// TwinCAT 3 PLC project PLC1_AssemblyLine
// Title: PLC1_AssemblyLine
// Company: Beckhoff Automation GmbH
// ProjectVersion: 1.0.0.0
// ProgramVersion: 3.1.4020.10
// libraries:
//   Tc2_MC2, * (Beckhoff Automation GmbH)
//   Tc2_Standard, * (Beckhoff Automation GmbH)
//   Tc2_System, * (Beckhoff Automation GmbH)
//   Tc3_EventLogger, * (Beckhoff Automation GmbH)
//   Tc3_Module, * (Beckhoff Automation GmbH)
// project tree:
//   DUTs/ E_FeederAutoState.TcDUT, E_AxisMode.TcDUT, E_StationState.TcDUT, ST_HmiAxisInfo.TcDUT, ST_HmiFeederInfo.TcDUT, ST_Hmi.TcDUT, ST_HmiAutomaticMode.TcDUT, ST_HmiErrorSimulation.TcDUT, ST_HmiFeederRecipe.TcDUT, ST_HmiManualMode.TcDUT, ST_HmiRecipeManagement.TcDUT, ST_PlcFeeder.TcDUT
//   GVLs/ GVL.TcGVL
//   / PlcTask.TcTTO
//   POUs/ FB_Axis.TcPOU, FB_Feeder.TcPOU, MAIN.TcPOU
//   Version/ Global_Version.TcGVL
// real-time tasks:
//   TASK PlcTask: cycle T#10ms, priority 10, ADS port 350
//   TASK Task 6: cycle T#10ms, priority 8, ADS port 301
// motion (NC):
//   TASK NC-Task-SAF: cycle T#2ms, priority 4, ADS port 501
//   TASK NC-Task-SVB: cycle T#10ms, priority 12, ADS port 511
//   AXIS Feeder1_AxisX (id 1)
//     OtherSettings: AllowMotionCmdToSlave=true
//     encoder EncType=1
//       SoftEndMinControl: Enable=true
//       SoftEndMaxControl: Enable=true, Range=5000
//     drive DrvType=5
//       TimeComp: TaskDelayCycles=1
//     controller CtrType=1
//       CtrPara: PriorControlFactor=1
//         Observer: BandWidth=20
//   AXIS Feeder1_AxisY (id 2)
//     OtherSettings: AllowMotionCmdToSlave=true
//     encoder EncType=1
//       SoftEndMinControl: Enable=true
//       SoftEndMaxControl: Enable=true, Range=5000
//     drive DrvType=5
//       TimeComp: TaskDelayCycles=1
//     controller CtrType=1
//       CtrPara: PriorControlFactor=1
//         Observer: BandWidth=20
//   AXIS Feeder2_AxisX (id 3)
//     OtherSettings: AllowMotionCmdToSlave=true
//     encoder EncType=1
//       SoftEndMinControl: Enable=true
//       SoftEndMaxControl: Enable=true, Range=5000
//     drive DrvType=5
//       TimeComp: TaskDelayCycles=1
//     controller CtrType=1
//       CtrPara: PriorControlFactor=1
//         Observer: BandWidth=20
//   AXIS Feeder2_AxisY (id 4)
//     OtherSettings: AllowMotionCmdToSlave=true
//     encoder EncType=1
//       SoftEndMinControl: Enable=true
//       SoftEndMaxControl: Enable=true, Range=5000
//     drive DrvType=5
//       TimeComp: TaskDelayCycles=1
//     controller CtrType=1
//       CtrPara: PriorControlFactor=1
//         Observer: BandWidth=20
// I/O:
//   DEVICE Gerät 3 (EtherCAT), AmsNetId 192.168.1.77.4.1
//     Klemme 1 (EK1100) [EK1100 EtherCAT-Koppler (2A E-Bus)]
//       Klemme 2 (EL1809) [EL1809 16K. Dig. Eingang 24V, 3ms]
//       Klemme 3 (EL2809) [EL2809 16K. Dig. Ausgang 24V, 0.5A]
//       Klemme 4 (EL9011) [EL9011 Endklemme]
// variable links:
//   PLC1_AssemblyLine/PLC1_AssemblyLine Instance <-> NC-Task-SAF/Axes/Feeder1_AxisX
//     PlcTask Inputs/MAIN.fbFeeder1.stPlcFeeder.fbAxisX.stAxis.NcToPlc <-> Outputs/ToPlc
//     PlcTask Outputs/MAIN.fbFeeder1.stPlcFeeder.fbAxisX.stAxis.PlcToNc <-> Inputs/FromPlc
//   PLC1_AssemblyLine/PLC1_AssemblyLine Instance <-> NC-Task-SAF/Axes/Feeder1_AxisY
//     PlcTask Inputs/MAIN.fbFeeder1.stPlcFeeder.fbAxisY.stAxis.NcToPlc <-> Outputs/ToPlc
//     PlcTask Outputs/MAIN.fbFeeder1.stPlcFeeder.fbAxisY.stAxis.PlcToNc <-> Inputs/FromPlc
//   PLC1_AssemblyLine/PLC1_AssemblyLine Instance <-> NC-Task-SAF/Axes/Feeder2_AxisX
//     PlcTask Inputs/MAIN.fbFeeder2.stPlcFeeder.fbAxisX.stAxis.NcToPlc <-> Outputs/ToPlc
//     PlcTask Outputs/MAIN.fbFeeder2.stPlcFeeder.fbAxisX.stAxis.PlcToNc <-> Inputs/FromPlc
//   PLC1_AssemblyLine/PLC1_AssemblyLine Instance <-> NC-Task-SAF/Axes/Feeder2_AxisY
//     PlcTask Inputs/MAIN.fbFeeder2.stPlcFeeder.fbAxisY.stAxis.NcToPlc <-> Outputs/ToPlc
//     PlcTask Outputs/MAIN.fbFeeder2.stPlcFeeder.fbAxisY.stAxis.PlcToNc <-> Inputs/FromPlc
//   Task 6 <-> Device 3 (EtherCAT)/Term 1 (EK1100)/Term 2 (EL1809)
//     Inputs/Var 1881 <-> Channel 1/Input

CONFIGURATION PLC1_AssemblyLine
    RESOURCE PLC ON TwinCAT3
        TASK PlcTask(INTERVAL := T#10ms, PRIORITY := 8);
        PROGRAM MAIN WITH PlcTask : MAIN;
    END_RESOURCE
END_CONFIGURATION

// ---- DUTs/E_FeederAutoState.TcDUT
{attribute 'qualified_only'}
TYPE E_FeederAutoState :
(
	eReset					:= 0,
	eMoveBackUp				:= 1,
	eMoveBackward			:= 2,
	eMoveDownForDragging	:= 3,
	eDrag					:= 4,
	eMoveUp					:= 5,
	eMoveForward			:= 6,
	eMoveDownForDropping	:= 7,
	eDrop					:= 8
);
END_TYPE

// ---- DUTs/E_AxisMode.TcDUT
{attribute 'qualified_only'}
TYPE E_AxisMode :
(
	INIT,
	ENABLE,
	JOG,
	POSITIONING,
	STOP,
	RESET,
	ERROR
);
END_TYPE

// ---- DUTs/E_StationState.TcDUT
{attribute 'qualified_only'}
TYPE E_StationState :
(
	eAuto	:= 2,
	eManual := 1,
	eStop	:= 0	
);
END_TYPE

// ---- DUTs/ST_HmiAxisInfo.TcDUT
TYPE ST_HmiAxisInfo :
STRUCT
	//Actual position
	fActPosition	: LREAL;
	//Actual velocity
	fActVelocity	: LREAL;
	//Current state of axis
	nAxisState		: UDINT;
	//Current mode of axis
	eAxisMode		: E_AxisMode;
END_STRUCT
END_TYPE

// ---- DUTs/ST_HmiFeederInfo.TcDUT
TYPE ST_HmiFeederInfo :
STRUCT
	//Bundled information about axis X
	stAxisX				: ST_HmiAxisInfo;
	
	//Bundled information about axis Y
	stAxisY				: ST_HmiAxisInfo;
	
	//Information about the gripper
	bGripperIsClosed	: BOOL;
END_STRUCT
END_TYPE

// ---- DUTs/ST_Hmi.TcDUT
TYPE ST_Hmi :
STRUCT
	//Operation mode 
	nStationState_Request	: INT;
	nStationState_Respond	: INT;	
	
	//Bundled manual mode settings and feedback
	stManualMode			: ST_HmiManualMode;
	
	//Bundled automatic mode settings and feedback
	stAutomaticMode			: ST_HmiAutomaticMode;
	
	//Bundled teach mode / recipe management settings and feedback
	stRecipeManagement		: ST_HmiRecipeManagement;
	
	//Bundled error simulation
	stErrorSimulation		: ST_HmiErrorSimulation;
	
	//Bundled feeder information
	stFeederInfo			: ST_HmiFeederInfo;
END_STRUCT
END_TYPE

// ---- DUTs/ST_HmiAutomaticMode.TcDUT
TYPE ST_HmiAutomaticMode :
STRUCT
	//Current state of the automatic mode state machine
	nStateNumber		: INT := 0;
END_STRUCT
END_TYPE

// ---- DUTs/ST_HmiErrorSimulation.TcDUT
TYPE ST_HmiErrorSimulation :
STRUCT
	bOnMoveBackUp			: BOOL;
	bOnMoveBackward			: BOOL;
	bOnMoveDownForDragging	: BOOL;
	bOnDrag					: BOOL;
	bOnMoveUp				: BOOL;
	bOnMoveForward			: BOOL;
	bOnMoveDownForDropping	: BOOL;
	bOnDrop					: BOOL;
END_STRUCT
END_TYPE

// ---- DUTs/ST_HmiFeederRecipe.TcDUT
TYPE ST_HmiFeederRecipe :
STRUCT
	//Target 1 name
	sTarget1Name			: STRING := 'Target Pos1';
	//Target 1 positon for X axis
	fTarget1PositionX		: LREAL	:= LREAL#0.0;
	//Target 1 position for Y axis
	fTarget1PositionY		: LREAL	:= LREAL#0.0;

	//Target 2 name
	sTarget2Name			: STRING := 'Target Pos2';
	//Target 2 positon for X axis
	fTarget2PositionX		: LREAL	:= LREAL#1000.0;
	//Target 2 position for Y axis
	fTarget2PositionY		: LREAL	:= LREAL#2000.0;
	
	//Velocity of both axis	
	fVelocity				: LREAL := 500;
END_STRUCT
END_TYPE

// ---- DUTs/ST_HmiManualMode.TcDUT
TYPE ST_HmiManualMode :
STRUCT
	//Manual mode - move X axis forward
	bButtonForwardX			: BOOL;
	//Manual mode - move X axis backward
	bButtonBackwardX		: BOOL;
	//Manual mode - move Y axis forward
	bButtonForwardY		: BOOL;
	//Manual mode - move Y axis backward
	bButtonBackwardY		: BOOL;
	//Manual mode - close gripper
	bButtonCloseGripper		: BOOL;
	//Manual mode - velocity X axis	
	fVelocityX			: LREAL := 500;
	//Manual mode - velocity Y axis
	fVelocityY			: LREAL := 500;
END_STRUCT
END_TYPE

// ---- DUTs/ST_HmiRecipeManagement.TcDUT
TYPE ST_HmiRecipeManagement :
STRUCT
	//Current recipe name
	sCurrentRecipeName	: STRING(50)	:= 'Unknown recipe';

	//Feeder recipe data
	stFeederRecipe		: ST_HmiFeederRecipe;
END_STRUCT
END_TYPE

// ---- DUTs/ST_PlcFeeder.TcDUT
TYPE ST_PlcFeeder :
STRUCT
	//ID of the feeder as identification in hmi, log, etc.
	nFeederId				: USINT;

	//Current operation mode of the machine
	eStationState			: E_StationState;
	
	//Delay for simulating drag and drop
	fbTonAuto				: TON;
	
	//State machine of automatic mode
	eAutoState				: E_FeederAutoState;

	//NC-drive X axis
	fbAxisX					: FB_Axis;
	//NC-drive Y axis
	fbAxisY					: FB_Axis;	

	//Gripper status
	bCloseGripper			: BOOL;
	bGripperIsClosed		: BOOL;
	
	//Current position of the X axis for historize extension in the HMI server
	fHmiPosXHistorize		: LREAL;
	//Current position of the Y axis for historize extension in the HMI server
	fHmiPosYHistorize		: LREAL;
	//Current velocity of the X axis for historize extension in the HMI server
	fHmiVeloXHistorize		: LREAL;
	//Current velocity of the Y axis for historize extension in the HMI server
	fHmiVeloYHistorize		: LREAL;
	
END_STRUCT
END_TYPE

// ---- GVLs/GVL.TcGVL
{attribute 'qualified_only'}
VAR_GLOBAL
	bAxisError	: BOOL;
END_VAR

// ---- Version/Global_Version.TcGVL
{attribute 'TcGenerated'}
// This function has been automatically generated from the project information.
VAR_GLOBAL CONSTANT
	{attribute 'const_non_replaced'}
	{attribute 'linkalways'}
	stLibVersion_PLC1_AssemblyLine : ST_LibVersion := (iMajor := 1, iMinor := 0, iBuild := 0, iRevision := 0, sVersion := '1.0.0.0');
END_VAR

// ---- POUs/MAIN.TcPOU
PROGRAM MAIN
VAR
	fbFeeder1		: FB_Feeder(nFeederId := 1);
	fbFeeder2		: FB_Feeder(nFeederId := 2);
END_VAR

fbFeeder1();
fbFeeder2();

END_PROGRAM

// ---- POUs/FB_Feeder.TcPOU
FUNCTION_BLOCK FB_Feeder
VAR_INPUT
END_VAR
VAR_OUTPUT
END_VAR
VAR
	
	stPlcFeeder				: ST_PlcFeeder;
	
	//Struct for communication with the HMI
	stHmi					: ST_Hmi;
END_VAR
VAR PERSISTENT
	//Current target positions from hmi recipe management
	stTargets				: ST_HmiFeederRecipe;
END_VAR

// Drives
stPlcFeeder.fbAxisX();
stPlcFeeder.fbAxisY();

// Hmi
M_Hmi();

// state machine
M_StationState();

// Events
M_Events();

CASE stHmi.nStationState_Request OF
	0: stPlcFeeder.eStationState := E_StationState.eStop;
	1: stPlcFeeder.eStationState := E_StationState.eManual;
	2: stPlcFeeder.eStationState := E_StationState.eAuto;
END_CASE

METHOD FB_init : BOOL
VAR_INPUT
	bInitRetains	: BOOL; // if TRUE, the retain variables are initialized (warm start / cold start)
	bInCopyCode		: BOOL;  // if TRUE, the instance afterwards gets moved into the copy code (online change)
	nFeederId		: USINT;
END_VAR
FeederId := nFeederId;
END_METHOD

PROPERTY PUBLIC FeederId : USINT
GET // PUBLIC
FeederId := stPlcFeeder.nFeederId;
END_GET
SET // PRIVATE
stPlcFeeder.nFeederId := FeederId;
END_SET
END_PROPERTY

METHOD M_Auto
VAR_INPUT
END_VAR
// Stoppping all axis for op mode change
IF stHmi.nStationState_Request <> 2 THEN
	stPlcFeeder.fbAxisX.bInStop := TRUE;
	stPlcFeeder.fbAxisY.bInStop := TRUE;
	RETURN;
END_IF

stPlcFeeder.fbTonAuto();
stPlcFeeder.fbAxisX.fInOverride := LREAL#100;    
stPlcFeeder.fbAxisX.fInVelocity := stTargets.fVelocity;
stPlcFeeder.fbAxisY.fInOverride := LREAL#100;    
stPlcFeeder.fbAxisY.fInVelocity := stTargets.fVelocity;

// State machine automatic mode
CASE stPlcFeeder.eAutoState OF
	E_FeederAutoState.eReset:
		M_AutoReset();
	E_FeederAutoState.eMoveBackUp:
		M_AutoMoveBackUp();
	E_FeederAutoState.eMoveBackward:
		M_AutoMoveBackward();	
	E_FeederAutoState.eMoveDownForDragging:
		M_AutoMoveDownForDragging();
	E_FeederAutoState.eDrag:
		M_AutoDrag();
	E_FeederAutoState.eMoveUp:
		M_AutoMoveUp();
	E_FeederAutoState.eMoveForward:
		M_AutoMoveForward();
	E_FeederAutoState.eMoveDownForDropping:
		M_AutoMoveDownForDropping();
	E_FeederAutoState.eDrop:
		M_AutoDrop();	
END_CASE
END_METHOD

METHOD M_AutoDrag
VAR_INPUT
END_VAR
VAR_INST
	fbAlarm						: Tc3_EventLogger.FB_TcAlarm;
	bWaitForErrorConfirmation	: BOOL;
	bConfirmManualy				: BOOL;
END_VAR
IF stHmi.stErrorSimulation.bOnDrag THEN
	fbAlarm.CreateEx(TC_EVENTS.AssemblyLineEvents.AutomaticModeError, TRUE, 0);
	fbAlarm.ipArguments.Clear().AddInt(stPlcFeeder.eAutoState);
END_IF

IF NOT bWaitForErrorConfirmation THEN
	stPlcFeeder.fbTonAuto.PT := T#2S;
	stPlcFeeder.fbTonAuto.IN := TRUE;
	stPlcFeeder.bCloseGripper := TRUE;
END_IF

IF stPlcFeeder.fbTonAuto.Q THEN
	stPlcFeeder.fbTonAuto.IN := FALSE;
	IF stHmi.stErrorSimulation.bOnDrag THEN
		stHmi.stErrorSimulation.bOnDrag := FALSE;		
		fbAlarm.Raise(0);
		bWaitForErrorConfirmation := TRUE;
	ELSE
		stPlcFeeder.bGripperIsClosed := TRUE;
		stPlcFeeder.eAutoState := E_FeederAutoState.eMoveUp;
	END_IF		
END_IF

IF bWaitForErrorConfirmation AND fbAlarm.eConfirmationState = TcEventConfirmationState.Confirmed THEN
	bWaitForErrorConfirmation := FALSE;
	fbAlarm.Clear(0,TRUE);	
	stPlcFeeder.bGripperIsClosed := TRUE;
	stPlcFeeder.eAutoState := E_FeederAutoState.eMoveUp;
END_IF

IF bConfirmManualy THEN
	bConfirmManualy := FALSE;
	fbAlarm.Confirm(0);
END_IF
END_METHOD

METHOD M_AutoDrop
VAR_INPUT
END_VAR
VAR_INST
	fbAlarm						: Tc3_EventLogger.FB_TcAlarm;
	bWaitForErrorConfirmation	: BOOL;
	bConfirmManualy				: BOOL;
END_VAR
IF stHmi.stErrorSimulation.bOnDrop THEN
	fbAlarm.CreateEx(TC_EVENTS.AssemblyLineEvents.AutomaticModeError, TRUE, 0);
	fbAlarm.ipArguments.Clear().AddInt(stPlcFeeder.eAutoState);
END_IF

IF NOT bWaitForErrorConfirmation THEN
	stPlcFeeder.fbTonAuto.PT := T#2S;
	stPlcFeeder.fbTonAuto.IN := TRUE;
	stPlcFeeder.bCloseGripper := FALSE;
END_IF

IF stPlcFeeder.fbTonAuto.Q THEN
	stPlcFeeder.fbTonAuto.IN := FALSE;
	IF stHmi.stErrorSimulation.bOnDrop THEN
		stHmi.stErrorSimulation.bOnDrop := FALSE;		
		fbAlarm.Raise(0);
		bWaitForErrorConfirmation := TRUE;
	ELSE
		stPlcFeeder.bGripperIsClosed := FALSE;
		stPlcFeeder.eAutoState := E_FeederAutoState.eMoveBackUp;
	END_IF		
END_IF

IF bWaitForErrorConfirmation AND fbAlarm.eConfirmationState = TcEventConfirmationState.Confirmed THEN
	bWaitForErrorConfirmation := FALSE;	
	fbAlarm.Clear(0,TRUE);
	stPlcFeeder.bGripperIsClosed := FALSE;
	stPlcFeeder.eAutoState := E_FeederAutoState.eMoveBackUp;
END_IF

IF bConfirmManualy THEN
	bConfirmManualy := FALSE;
	fbAlarm.Confirm(0);
END_IF
END_METHOD

METHOD M_AutoMoveBackUp
VAR_INPUT
END_VAR
VAR_INST
	fbAlarm						: Tc3_EventLogger.FB_TcAlarm;
	bWaitForErrorConfirmation	: BOOL;
	bConfirmManualy				: BOOL;
END_VAR
IF stHmi.stErrorSimulation.bOnMoveBackUp THEN
	fbAlarm.CreateEx(TC_EVENTS.AssemblyLineEvents.AutomaticModeError, TRUE, 0);
	fbAlarm.ipArguments.Clear().AddInt(stPlcFeeder.eAutoState);
END_IF

stPlcFeeder.fbAxisY.fInTargetPos := 0.0;

IF stPlcFeeder.fbAxisY.fOutActPosition <> 0 THEN
	stPlcFeeder.fbAxisY.bInPositioning := TRUE;
	IF stHmi.stErrorSimulation.bOnMoveBackUp THEN
		stHmi.stErrorSimulation.bOnMoveBackUp := FALSE;
		stPlcFeeder.fbAxisX.bInPositioning := FALSE;		
		stPlcFeeder.fbAxisY.bInPositioning := FALSE;		
		stPlcFeeder.fbAxisX.bInStop := TRUE;
		stPlcFeeder.fbAxisY.bInStop := TRUE;
		fbAlarm.Raise(0);
		bWaitForErrorConfirmation := TRUE;
	END_IF
ELSIF stPlcFeeder.fbAxisY.fOutActPosition = 0 AND NOT bWaitForErrorConfirmation THEN 
	stPlcFeeder.fbAxisY.bInPositioning := FALSE;
	stPlcFeeder.eAutoState :=  E_FeederAutoState.eMoveBackward;
END_IF

IF bWaitForErrorConfirmation AND fbAlarm.eConfirmationState = TcEventConfirmationState.Confirmed THEN
	bWaitForErrorConfirmation := FALSE;	
	fbAlarm.Clear(0,TRUE);
	stPlcFeeder.fbAxisX.bInStop := FALSE;
	stPlcFeeder.fbAxisY.bInStop := FALSE;
	stPlcFeeder.fbAxisY.bInPositioning := TRUE;
END_IF

IF bConfirmManualy THEN
	bConfirmManualy := FALSE;
	fbAlarm.Confirm(0);
END_IF
END_METHOD

METHOD M_AutoMoveBackward
VAR_INPUT
END_VAR
VAR_INST
	fbAlarm						: Tc3_EventLogger.FB_TcAlarm;
	bWaitForErrorConfirmation	: BOOL;
	bConfirmManualy				: BOOL;
END_VAR
IF stHmi.stErrorSimulation.bOnMoveBackward THEN
	fbAlarm.CreateEx(TC_EVENTS.AssemblyLineEvents.AutomaticModeError, TRUE, 0);
	fbAlarm.ipArguments.Clear().AddInt(stPlcFeeder.eAutoState);
END_IF

stPlcFeeder.fbAxisX.fInTargetPos := stTargets.fTarget1PositionX;

IF stPlcFeeder.fbAxisX.fOutActPosition <> stTargets.fTarget1PositionX THEN
	stPlcFeeder.fbAxisX.bInPositioning := TRUE;
	IF stHmi.stErrorSimulation.bOnMoveBackward THEN
		stHmi.stErrorSimulation.bOnMoveBackward := FALSE;
		stPlcFeeder.fbAxisX.bInPositioning := FALSE;		
		stPlcFeeder.fbAxisY.bInPositioning := FALSE;		
		stPlcFeeder.fbAxisX.bInStop := TRUE;
		stPlcFeeder.fbAxisY.bInStop := TRUE;
		fbAlarm.Raise(0);
		bWaitForErrorConfirmation := TRUE;
	END_IF
ELSIF stPlcFeeder.fbAxisX.fOutActPosition = stTargets.fTarget1PositionX AND NOT bWaitForErrorConfirmation THEN 
	stPlcFeeder.fbAxisX.bInPositioning := FALSE;
	stPlcFeeder.eAutoState := E_FeederAutoState.eMoveDownForDragging;
END_IF

IF bWaitForErrorConfirmation AND fbAlarm.eConfirmationState = TcEventConfirmationState.Confirmed THEN
	bWaitForErrorConfirmation := FALSE;	
	fbAlarm.Clear(0,TRUE);	
	stPlcFeeder.fbAxisX.bInStop := FALSE;
	stPlcFeeder.fbAxisY.bInStop := FALSE;
	stPlcFeeder.fbAxisX.bInPositioning := TRUE;
END_IF

IF bConfirmManualy THEN
	bConfirmManualy := FALSE;
	fbAlarm.Confirm(0);
END_IF
END_METHOD

METHOD M_AutoMoveDownForDragging
VAR_INPUT
END_VAR
VAR_INST
	fbAlarm						: Tc3_EventLogger.FB_TcAlarm;
	bWaitForErrorConfirmation	: BOOL;
	bConfirmManualy				: BOOL;
END_VAR
IF stHmi.stErrorSimulation.bOnMoveDownForDragging THEN
	fbAlarm.CreateEx(TC_EVENTS.AssemblyLineEvents.AutomaticModeError, TRUE, 0);
	fbAlarm.ipArguments.Clear().AddInt(stPlcFeeder.eAutoState);
END_IF

stPlcFeeder.fbAxisY.fInTargetPos := stTargets.fTarget1PositionY;

IF stPlcFeeder.fbAxisY.fOutActPosition <> stTargets.fTarget1PositionY THEN
	stPlcFeeder.fbAxisY.bInPositioning := TRUE;
	IF stHmi.stErrorSimulation.bOnMoveDownForDragging THEN
		stHmi.stErrorSimulation.bOnMoveDownForDragging := FALSE;
		stPlcFeeder.fbAxisX.bInPositioning := FALSE;		
		stPlcFeeder.fbAxisY.bInPositioning := FALSE;		
		stPlcFeeder.fbAxisX.bInStop := TRUE;
		stPlcFeeder.fbAxisY.bInStop := TRUE;
		fbAlarm.Raise(0);
		bWaitForErrorConfirmation := TRUE;
	END_IF
ELSIF stPlcFeeder.fbAxisY.fOutActPosition = stTargets.fTarget1PositionY AND NOT bWaitForErrorConfirmation THEN 
	stPlcFeeder.fbAxisY.bInPositioning := FALSE;
	stPlcFeeder.eAutoState := E_FeederAutoState.eDrag;
END_IF

IF bWaitForErrorConfirmation AND fbAlarm.eConfirmationState = TcEventConfirmationState.Confirmed THEN
	bWaitForErrorConfirmation := FALSE;	
	fbAlarm.Clear(0,TRUE);
	stPlcFeeder.fbAxisX.bInStop := FALSE;
	stPlcFeeder.fbAxisY.bInStop := FALSE;
	stPlcFeeder.fbAxisY.bInPositioning := TRUE;
END_IF

IF bConfirmManualy THEN
	bConfirmManualy := FALSE;
	fbAlarm.Confirm(0);
END_IF
END_METHOD

METHOD M_AutoMoveDownForDropping
VAR_INPUT
END_VAR
VAR_INST
	fbAlarm						: Tc3_EventLogger.FB_TcAlarm;
	bWaitForErrorConfirmation	: BOOL;
	bConfirmManualy				: BOOL;
END_VAR
IF stHmi.stErrorSimulation.bOnMoveDownForDropping THEN
	fbAlarm.CreateEx(TC_EVENTS.AssemblyLineEvents.AutomaticModeError, TRUE, 0);
	fbAlarm.ipArguments.Clear().AddInt(stPlcFeeder.eAutoState);
END_IF

stPlcFeeder.fbAxisY.fInTargetPos := stTargets.fTarget2PositionY;

IF stPlcFeeder.fbAxisY.fOutActPosition <> stTargets.fTarget2PositionY THEN
	stPlcFeeder.fbAxisY.bInPositioning := TRUE;
	IF stHmi.stErrorSimulation.bOnMoveDownForDropping THEN
		stHmi.stErrorSimulation.bOnMoveDownForDropping := FALSE;
		stPlcFeeder.fbAxisX.bInPositioning := FALSE;		
		stPlcFeeder.fbAxisY.bInPositioning := FALSE;		
		stPlcFeeder.fbAxisX.bInStop := TRUE;
		stPlcFeeder.fbAxisY.bInStop := TRUE;
		fbAlarm.Raise(0);
		bWaitForErrorConfirmation := TRUE;
	END_IF
ELSIF stPlcFeeder.fbAxisY.fOutActPosition = stTargets.fTarget2PositionY AND NOT bWaitForErrorConfirmation THEN 
	stPlcFeeder.fbAxisY.bInPositioning := FALSE;
	stPlcFeeder.eAutoState := E_FeederAutoState.eDrop;
END_IF

IF bWaitForErrorConfirmation AND fbAlarm.eConfirmationState = TcEventConfirmationState.Confirmed THEN
	bWaitForErrorConfirmation := FALSE;	
	fbAlarm.Clear(0,TRUE);
	stPlcFeeder.fbAxisX.bInStop := FALSE;
	stPlcFeeder.fbAxisY.bInStop := FALSE;
	stPlcFeeder.fbAxisY.bInPositioning := TRUE;
END_IF

IF bConfirmManualy THEN
	bConfirmManualy := FALSE;
	fbAlarm.Confirm(0);
END_IF
END_METHOD

METHOD M_AutoMoveForward
VAR_INPUT
END_VAR
VAR_INST
	fbAlarm						: Tc3_EventLogger.FB_TcAlarm;
	bWaitForErrorConfirmation	: BOOL;
	bConfirmManualy				: BOOL;
END_VAR
IF stHmi.stErrorSimulation.bOnMoveForward THEN
	fbAlarm.CreateEx(TC_EVENTS.AssemblyLineEvents.AutomaticModeError, TRUE, 0);
	fbAlarm.ipArguments.Clear().AddInt(stPlcFeeder.eAutoState);
END_IF

stPlcFeeder.fbAxisX.fInTargetPos := stTargets.fTarget2PositionX;

IF stPlcFeeder.fbAxisX.fOutActPosition <> stTargets.fTarget2PositionX THEN
	stPlcFeeder.fbAxisX.bInPositioning := TRUE;
	IF stHmi.stErrorSimulation.bOnMoveForward THEN
		stHmi.stErrorSimulation.bOnMoveForward := FALSE;
		stPlcFeeder.fbAxisX.bInPositioning := FALSE;		
		stPlcFeeder.fbAxisY.bInPositioning := FALSE;		
		stPlcFeeder.fbAxisX.bInStop := TRUE;
		stPlcFeeder.fbAxisY.bInStop := TRUE;
		fbAlarm.Raise(0);
		bWaitForErrorConfirmation := TRUE;
	END_IF
ELSIF stPlcFeeder.fbAxisX.fOutActPosition = stTargets.fTarget2PositionX AND NOT bWaitForErrorConfirmation THEN 
	stPlcFeeder.fbAxisX.bInPositioning := FALSE;
	stPlcFeeder.eAutoState := E_FeederAutoState.eMoveDownForDropping;
END_IF

IF bWaitForErrorConfirmation AND fbAlarm.eConfirmationState = TcEventConfirmationState.Confirmed THEN
	bWaitForErrorConfirmation := FALSE;	
	fbAlarm.Clear(0,TRUE);
	stPlcFeeder.fbAxisX.bInStop := FALSE;
	stPlcFeeder.fbAxisY.bInStop := FALSE;
	stPlcFeeder.fbAxisX.bInPositioning := TRUE;
END_IF

IF bConfirmManualy THEN
	bConfirmManualy := FALSE;
	fbAlarm.Confirm(0);
END_IF
END_METHOD

METHOD M_AutoMoveUp
VAR_INPUT
END_VAR
VAR_INST
	fbAlarm						: Tc3_EventLogger.FB_TcAlarm;
	bWaitForErrorConfirmation	: BOOL;
	bConfirmManualy				: BOOL;
END_VAR
IF stHmi.stErrorSimulation.bOnMoveUp THEN
	fbAlarm.CreateEx(TC_EVENTS.AssemblyLineEvents.AutomaticModeError, TRUE, 0);
	fbAlarm.ipArguments.Clear().AddInt(stPlcFeeder.eAutoState);
END_IF

stPlcFeeder.fbAxisY.fInTargetPos := 0.0;

IF stPlcFeeder.fbAxisY.fOutActPosition <> 0 THEN
	stPlcFeeder.fbAxisY.bInPositioning := TRUE;
	IF stHmi.stErrorSimulation.bOnMoveUp THEN
		stHmi.stErrorSimulation.bOnMoveUp := FALSE;
		stPlcFeeder.fbAxisX.bInPositioning := FALSE;		
		stPlcFeeder.fbAxisY.bInPositioning := FALSE;		
		stPlcFeeder.fbAxisX.bInStop := TRUE;
		stPlcFeeder.fbAxisY.bInStop := TRUE;
		fbAlarm.Raise(0);
		bWaitForErrorConfirmation := TRUE;
	END_IF
ELSIF stPlcFeeder.fbAxisY.fOutActPosition = 0 AND NOT bWaitForErrorConfirmation THEN 
	stPlcFeeder.fbAxisY.bInPositioning := FALSE;
	stPlcFeeder.eAutoState := E_FeederAutoState.eMoveForward;
END_IF

IF bWaitForErrorConfirmation AND fbAlarm.eConfirmationState = TcEventConfirmationState.Confirmed THEN
	bWaitForErrorConfirmation := FALSE;	
	fbAlarm.Clear(0,TRUE);
	stPlcFeeder.fbAxisX.bInStop := FALSE;
	stPlcFeeder.fbAxisY.bInStop := FALSE;
	stPlcFeeder.fbAxisY.bInPositioning := TRUE;
END_IF

IF bConfirmManualy THEN
	bConfirmManualy := FALSE;
	fbAlarm.Confirm(0);
END_IF
END_METHOD

METHOD M_AutoReset
VAR_INPUT
END_VAR
stPlcFeeder.fbAxisX.fInTargetPos := 0.0;
stPlcFeeder.fbAxisY.fInTargetPos := 0.0;
stPlcFeeder.fbAxisX.bInStop := FALSE;
stPlcFeeder.fbAxisY.bInStop := FALSE;

IF stPlcFeeder.fbAxisX.fOutActPosition <> 0 THEN 
	stPlcFeeder.fbAxisX.bInPositioning := TRUE;
END_IF

IF stPlcFeeder.fbAxisY.fOutActPosition <> 0 THEN 
	stPlcFeeder.fbAxisY.bInPositioning := TRUE;
END_IF

IF stPlcFeeder.fbAxisX.fOutActPosition = 0 AND stPlcFeeder.fbAxisY.fOutActPosition = 0 THEN 
	stPlcFeeder.fbAxisX.bInPositioning := FALSE;
	stPlcFeeder.fbAxisY.bInPositioning := FALSE;
	stPlcFeeder.eAutoState := E_FeederAutoState.eMoveBackUp;
END_IF
END_METHOD

METHOD PRIVATE M_Events : BOOL
VAR_INPUT
END_VAR
VAR
	sJsonAttributeAxis		: STRING;
END_VAR
VAR_INST
	fbTriggerAutomaticOn	: R_TRIG;
	fbTriggerManualModeOn	: R_TRIG;
	fbTriggerStop			: R_TRIG;
	fbTriggerErrorAxisX		: R_TRIG;
	fbTriggerErrorAxisY		: R_TRIG;	
	fbMessage 				: Tc3_EventLogger.FB_TcMessage;
	fbAlarmAxisX			: Tc3_EventLogger.FB_TcAlarm;
	fbAlarmAxisY			: Tc3_EventLogger.FB_TcAlarm;
END_VAR
fbTriggerAutomaticOn(CLK := stPlcFeeder.eStationState = E_StationState.eAuto);
IF fbTriggerAutomaticOn.Q THEN
	fbMessage.CreateEx(TC_EVENTS.AssemblyLineEvents.FeederAutomaticOn, 0);
	fbMessage.ipArguments.Clear().AddUSInt(FeederId);
	fbMessage.Send(0);
END_IF

fbTriggerManualModeOn(CLK := stPlcFeeder.eStationState = E_StationState.eManual);
IF fbTriggerManualModeOn.Q THEN
	fbMessage.CreateEx(TC_EVENTS.AssemblyLineEvents.FeederManualModeOn, 0);
	fbMessage.ipArguments.Clear().AddUSInt(FeederId);
	fbMessage.Send(0);
END_IF

fbTriggerStop(CLK := stPlcFeeder.eStationState = E_StationState.eStop);
IF fbTriggerStop.Q THEN
	fbMessage.CreateEx(TC_EVENTS.AssemblyLineEvents.FeederStopped, 0);
	fbMessage.ipArguments.Clear().AddUSInt(FeederId);
	fbMessage.Send(0);
END_IF

fbTriggerErrorAxisX(CLK := stPlcFeeder.fbAxisX.bOutError);
IF fbTriggerErrorAxisX.Q THEN
	fbAlarmAxisX.Clear(0, TRUE);
	fbAlarmAxisX.CreateEx(TC_EVENTS.AssemblyLineEvents.FeederError, FALSE, 0);
	fbAlarmAxisX.ipArguments.Clear().AddUSInt(FeederId).AddString('X');
	sJsonAttributeAxis := CONCAT(CONCAT('{"ErrorId: ', TO_STRING(stPlcFeeder.fbAxisX.nOutErrorId)), '}');
	fbAlarmAxisX.SetJsonAttribute(sJsonAttributeAxis);
	fbAlarmAxisX.Raise(0);
END_IF

fbTriggerErrorAxisY(CLK := stPlcFeeder.fbAxisY.bOutError);
IF fbTriggerErrorAxisY.Q THEN
	fbAlarmAxisY.Clear(0, TRUE);
	fbAlarmAxisY.CreateEx(TC_EVENTS.AssemblyLineEvents.FeederError, FALSE, 0);
	fbAlarmAxisY.ipArguments.Clear().AddUSInt(FeederId).AddString('Y');
	sJsonAttributeAxis := CONCAT(CONCAT('{"ErrorId: ', TO_STRING(stPlcFeeder.fbAxisY.nOutErrorId)), '}');
	fbAlarmAxisY.SetJsonAttribute(sJsonAttributeAxis);
	fbAlarmAxisY.Raise(0);
END_IF
END_METHOD

METHOD M_Hmi : BOOL
VAR_INPUT
END_VAR
IF _TaskInfo[GETCURTASKINDEXEX()].FirstCycle THEN
	stHmi.stRecipeManagement.stFeederRecipe := stTargets;
END_IF

stHmi.nStationState_Respond := TO_INT(stPlcFeeder.eStationState);

stHmi.stAutomaticMode.nStateNumber := stPlcFeeder.eAutoState;
stHmi.stFeederInfo.bGripperIsClosed := stPlcFeeder.bGripperIsClosed;

// HMI historize actual position and velocity
stPlcFeeder.fHmiPosXHistorize := stPlcFeeder.fbAxisX.fOutActPosition;
stPlcFeeder.fHmiPosYHistorize := stPlcFeeder.fbAxisY.fOutActPosition;
stPlcFeeder.fHmiVeloXHistorize := stPlcFeeder.fbAxisX.fOutActVelocity;
stPlcFeeder.fHmiVeloYHistorize := stPlcFeeder.fbAxisY.fOutActVelocity;

// HMI axis information
stHmi.stFeederInfo.stAxisX.fActPosition := stPlcFeeder.fbAxisX.fOutActPosition;
stHmi.stFeederInfo.stAxisX.fActVelocity := stPlcFeeder.fbAxisX.fOutActVelocity;
stHmi.stFeederInfo.stAxisX.nAxisState := stPlcFeeder.fbAxisX.nOutAxisState;
stHmi.stFeederInfo.stAxisX.eAxisMode := stPlcFeeder.fbAxisX.eOutAxisMode;

stHmi.stFeederInfo.stAxisY.fActPosition := stPlcFeeder.fbAxisY.fOutActPosition;
stHmi.stFeederInfo.stAxisY.fActVelocity := stPlcFeeder.fbAxisY.fOutActVelocity;
stHmi.stFeederInfo.stAxisY.nAxisState := stPlcFeeder.fbAxisY.nOutAxisState;
stHmi.stFeederInfo.stAxisY.eAxisMode := stPlcFeeder.fbAxisY.eOutAxisMode;

//Set targets from hmi recipe management
stTargets := stHmi.stRecipeManagement.stFeederRecipe;
END_METHOD

METHOD M_Man
VAR_INPUT
END_VAR
// Stoppping all axis for op mode change
IF stHmi.nStationState_Request <> 1 THEN
	stPlcFeeder.fbAxisX.bInStop := TRUE;
	stPlcFeeder.fbAxisY.bInStop := TRUE;
	stPlcFeeder.fbAxisX.bInJog := FALSE;
	stPlcFeeder.fbAxisY.bInJog := FALSE;
	stPlcFeeder.eAutoState := E_FeederAutoState.eReset;
	RETURN;
END_IF

stPlcFeeder.fbAxisX.bInStop := FALSE;
stPlcFeeder.fbAxisX.bInJog := TRUE;
stPlcFeeder.fbAxisX.fInOverride := LREAL#100;
stPlcFeeder.fbAxisX.fInVelocity := stHmi.stManualMode.fVelocityX;
stPlcFeeder.fbAxisX.bInJogForward := stHmi.stManualMode.bButtonForwardX;
stPlcFeeder.fbAxisX.bInJogBackward := stHmi.stManualMode.bButtonBackwardX;

stPlcFeeder.fbAxisY.bInStop := FALSE;
stPlcFeeder.fbAxisY.bInJog := TRUE;
stPlcFeeder.fbAxisY.fInOverride := LREAL#100;
stPlcFeeder.fbAxisY.fInVelocity := stHmi.stManualMode.fVelocityY;
stPlcFeeder.fbAxisY.bInJogForward := stHmi.stManualMode.bButtonForwardY;
stPlcFeeder.fbAxisY.bInJogBackward := stHmi.stManualMode.bButtonBackwardY;

stPlcFeeder.bCloseGripper := stHmi.stManualMode.bButtonCloseGripper;
END_METHOD

METHOD M_StationState
VAR_INPUT
END_VAR

VAR

END_VAR
CASE stPlcFeeder.eStationState OF
	E_StationState.eAuto:
		M_Auto();
	E_StationState.eManual:
		M_Man();
	E_StationState.eStop:
		M_Stop();	
END_CASE
END_METHOD

METHOD M_Stop
VAR_INPUT
END_VAR
stPlcFeeder.fbAxisX.bInStop := TRUE;
stPlcFeeder.fbAxisY.bInStop := TRUE;

IF stHmi.nStationState_Request = 2 THEN
	stPlcFeeder.eAutoState := E_FeederAutoState.eReset;
END_IF
END_METHOD

END_FUNCTION_BLOCK

// ---- POUs/FB_Axis.TcPOU
FUNCTION_BLOCK FB_Axis
VAR_INPUT
	// Commands
	bInJog				: BOOL;
	bInJogForward		: BOOL;
	bInJogBackward		: BOOL;
	bInPositioning		: BOOL;
	bInStop				: BOOL;
	bInReset			: BOOL;

	// Parameters
	fInVelocity			: LREAL := 1000.0;
	fInOverride			: LREAL := 100;
	fInTargetPos		: LREAL := 0;	
END_VAR
VAR_OUTPUT
	// Status
	bOutError			: BOOL;
	nOutErrorId			: UDINT;
	fOutActPosition		: DINT;
	fOutActVelocity		: DINT;
	fOutSetPosition		: LREAL;
	fOutSetVelocity		: LREAL;
	nOutAxisState		: UDINT;
	eOutAxisMode		: E_AxisMode;    
END_VAR
VAR
	// MC function blocks
	fbPower			: Tc2_MC2.MC_Power;
	fbReset			: Tc2_MC2.MC_Reset;
	fbStop			: Tc2_MC2.MC_Stop;	
	fbMoveAbs		: Tc2_MC2.MC_MoveAbsolute;
	fbJog			: Tc2_MC2.MC_Jog;
	
	// MC structures	
	stAxis			: Tc2_MC2.AXIS_REF;
	stPower			: Tc2_MC2.ST_McOutputs;
	stReset			: Tc2_MC2.ST_McOutputs;
	stStop			: Tc2_MC2.ST_McOutputs;
	stMoveAbs		: Tc2_MC2.ST_McOutputs;
	stJog			: Tc2_MC2.ST_McOutputs;
	
	// state machine
	eAxisMode		: E_AxisMode;
END_VAR

stAxis.ReadStatus();

// state machine
CASE eAxisMode OF

		E_AxisMode.INIT:
		
					fbPower.Enable := FALSE;
					fbReset.Execute := FALSE;
					fbStop.Execute := FALSE;
					fbMoveAbs.Execute := FALSE;
					fbJog.JogForward := FALSE;
					fbJog.JogBackwards := FALSE;
					eAxisMode := E_AxisMode.ENABLE;		
					
		E_AxisMode.ENABLE:					

					fbPower.Enable := TRUE;
					fbPower.Enable_Positive := TRUE;
					fbPower.Enable_Negative := TRUE;
					
					IF fbPower.Status THEN
						IF  bInStop THEN
							eAxisMode := E_AxisMode.STOP;						
						ELSIF  bInJog THEN
							eAxisMode := E_AxisMode.JOG;
						ELSIF bInPositioning THEN
							eAxisMode := E_AxisMode.POSITIONING;
						ELSIF  bInReset THEN
							eAxisMode := E_AxisMode.RESET;
						END_IF
					ELSIF fbPower.Error THEN
						eAxisMode := E_AxisMode.ERROR;						
					END_IF
					
					bOutError := fbPower.Error;
					nOutErrorId := fbPower.ErrorID;

		E_AxisMode.JOG: // Jog / manual mode with continuous speed *)					
        
					fbJog.Mode := Tc2_MC2.MC_JOGMODE_CONTINOUS;
					fbJog.Velocity := fInVelocity;
					
					IF NOT bInStop THEN
						fbJog.JogForward := bInJogForward;
						fbJog.JogBackwards := bInJogBackward;					
					END_IF
					
					IF NOT bInJog THEN
						eAxisMode := E_AxisMode.STOP;
					END_IF 
					
					(* error state *)
					IF fbJog.Error THEN
						eAxisMode := E_AxisMode.ERROR;
					END_IF
					
					bOutError := fbJog.Error;
					nOutErrorId := fbJog.ErrorID;
		
		E_AxisMode.POSITIONING: // Positioning run
				
					IF bInPositioning AND NOT fbMoveAbs.Busy THEN
						fbMoveAbs.Velocity := fInVelocity;
						fbMoveAbs.Position := fInTargetPos;
						fbMoveAbs.Execute := TRUE;
					END_IF
					
					// Wait for postioning run done
					IF fbMoveAbs.Done OR bInStop THEN
						bInPositioning := FALSE;
						fbMoveAbs.Execute := FALSE;
						eAxisMode := E_AxisMode.STOP;
					END_IF
					
					// Check if axis has an error
					IF fbMoveAbs.Error THEN
						eAxisMode := E_AxisMode.ERROR;
					END_IF
					
					bOutError := fbMoveAbs.Error;
					nOutErrorId := fbMoveAbs.ErrorID;	
					
		E_AxisMode.STOP: (* stops axis from continuos motion *)				
					fbStop.Execute := TRUE;
					IF fbStop.Active THEN
						fbStop.Execute := FALSE;
						bInStop := FALSE;
						IF fbStop.Done THEN
							bInStop := FALSE;
							eAxisMode := E_AxisMode.ENABLE;
						END_IF
					END_IF
					
					(* error state *)
					IF fbStop.Error THEN
						eAxisMode := E_AxisMode.ERROR;
					END_IF
					
					bOutError := fbStop.Error;
					nOutErrorId := fbStop.ErrorID;	

		E_AxisMode.RESET: //Reset drive to take new motion commands			

					fbReset.Execute := TRUE;
					IF fbReset.Busy THEN
						fbReset.Execute := FALSE;
						bInReset:= FALSE;
					END_IF
					IF fbReset.Done THEN
						eAxisMode := E_AxisMode.INIT;
					ELSIF fbReset.Error THEN
						eAxisMode := E_AxisMode.ERROR;
					END_IF
					
					bOutError := fbReset.Error;
					nOutErrorId := fbReset.ErrorID;

		E_AxisMode.ERROR:					

					IF stAxis.Status.Error THEN
						eAxisMode := E_AxisMode.RESET;
					ELSE
						eAxisMode := E_AxisMode.INIT;
					END_IF				

END_CASE

// Call MC function blocks
Power();
Reset();
Stop();
MoveAbs();
Jog();

// Status outputs
fOutActVelocity := TO_DINT(stAxis.NcToPlc.ActVelo);
fOutActPosition := TO_DINT(stAxis.NcToPlc.ActPos);
fOutSetVelocity := TO_LREAL(TO_DINT(stAxis.NcToPlc.SetVelo * 10000)) / 10000;
fOutSetPosition := TO_LREAL(TO_DINT(stAxis.NcToPlc.SetPos * 10000)) / 10000;
nOutAxisState := stAxis.NcToPlc.AxisState;
eOutAxisMode := eAxisMode;

ACTION Jog:
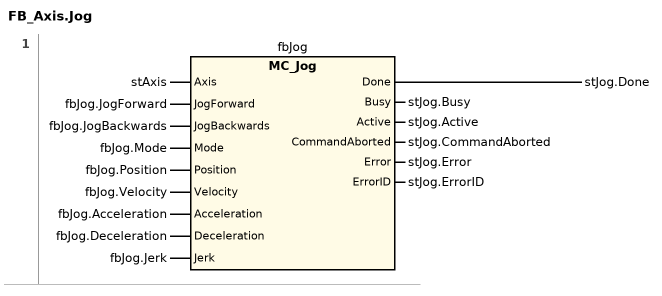
// NETWORK 1
fbJog(
    Axis := stAxis,
    JogForward := fbJog.JogForward,
    JogBackwards := fbJog.JogBackwards,
    Mode := fbJog.Mode,
    Position := fbJog.Position,
    Velocity := fbJog.Velocity,
    Acceleration := fbJog.Acceleration,
    Deceleration := fbJog.Deceleration,
    Jerk := fbJog.Jerk,
    Busy => stJog.Busy,
    Active => stJog.Active,
    CommandAborted => stJog.CommandAborted,
    Error => stJog.Error,
    ErrorID => stJog.ErrorID); // MC_Jog
stJog.Done := fbJog.Done;
END_ACTION

ACTION MoveAbs:
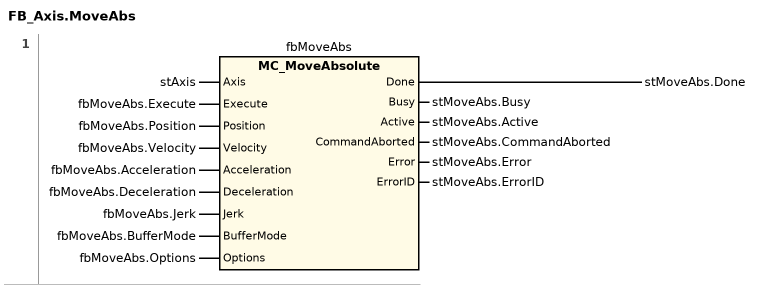
// NETWORK 1
fbMoveAbs(
    Axis := stAxis,
    Execute := fbMoveAbs.Execute,
    Position := fbMoveAbs.Position,
    Velocity := fbMoveAbs.Velocity,
    Acceleration := fbMoveAbs.Acceleration,
    Deceleration := fbMoveAbs.Deceleration,
    Jerk := fbMoveAbs.Jerk,
    BufferMode := fbMoveAbs.BufferMode,
    Options := fbMoveAbs.Options,
    Busy => stMoveAbs.Busy,
    Active => stMoveAbs.Active,
    CommandAborted => stMoveAbs.CommandAborted,
    Error => stMoveAbs.Error,
    ErrorID => stMoveAbs.ErrorID); // MC_MoveAbsolute
stMoveAbs.Done := fbMoveAbs.Done;
END_ACTION

ACTION Power:
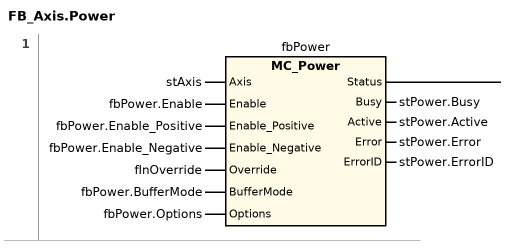
// NETWORK 1
fbPower(
    Axis := stAxis,
    Enable := fbPower.Enable,
    Enable_Positive := fbPower.Enable_Positive,
    Enable_Negative := fbPower.Enable_Negative,
    Override := fInOverride,
    BufferMode := fbPower.BufferMode,
    Options := fbPower.Options,
    Busy => stPower.Busy,
    Active => stPower.Active,
    Error => stPower.Error,
    ErrorID => stPower.ErrorID); // MC_Power
END_ACTION

ACTION Reset:
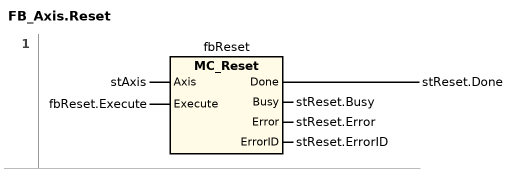
// NETWORK 1
fbReset(
    Axis := stAxis,
    Execute := fbReset.Execute,
    Busy => stReset.Busy,
    Error => stReset.Error,
    ErrorID => stReset.ErrorID); // MC_Reset
stReset.Done := fbReset.Done;
END_ACTION

ACTION Stop:
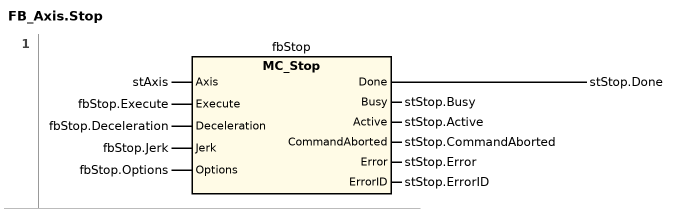
// NETWORK 1
fbStop(
    Axis := stAxis,
    Execute := fbStop.Execute,
    Deceleration := fbStop.Deceleration,
    Jerk := fbStop.Jerk,
    Options := fbStop.Options,
    Busy => stStop.Busy,
    Active => stStop.Active,
    CommandAborted => stStop.CommandAborted,
    Error => stStop.Error,
    ErrorID => stStop.ErrorID); // MC_Stop
stStop.Done := fbStop.Done;
END_ACTION

END_FUNCTION_BLOCK
